FUNCTION_BLOCK Q_SoftKeyMask (* Command change soft key mask( Part 6 - F.36 ) *)
  (* Standard: ISO 11783-6; Description: Copyright (c) 2022 HR Agrartechnik GmbH This program and the accompanying materials are made available under the terms of the Eclipse Public License 2.0 which is available at https://www.eclipse.org/legal/epl-2.0/ SPDX-License-Identifier: EPL-2.0 see Description Tab *)
  (* Version 1.0, 2022-07-08, Franz Höpfinger, HR Agrartechnik GmbH *)
  (* Documentation:
  Command change soft key mask( Part 6 - F.36 )
   This command is used to change the soft key mask associated with a data or alarm mask object.
   param[in] {type, uint8_t}
   1 == Data, 2 == Alarm
   param[in] {dataOrAlarmMaskObjectID, uint16_t}
   Object ID of active Mask
   param[in] {newSoftKeyMaskObjectID, uint16_t}
   Object ID of (new) soft key mask
   Return Values: 
   int16_t
    - VT_E_NO_ERR (0) - OK
   - VT_E_OVERFLOW (-6) - buffer overflow
   - VT_E_NOACT (-8) - Command not possible in current state
   - VT_E_NO_INSTANCE (-21) - No VT client available
   - VT_E_ISO_INSTANCE_INVALID (-129) - Identifier for instance (connection) invalid
   - VT_E_NOT_ALIVE (-130) - Identifier for instance valid, but VT Dead.
  *)
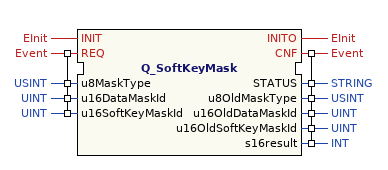
  EVENT_INPUT
    INIT : EInit; (* Service Initialization *)
    REQ WITH u16DataMaskId, u16SoftKeyMaskId, u8MaskType; (* Service Request *)
  END_EVENT
  EVENT_OUTPUT
    INITO : EInit; (* Initialization Confirm *)
    CNF WITH STATUS, s16result, u16OldDataMaskId, u16OldSoftKeyMaskId, u8OldMaskType; (* Confirmation of Requested Service *)
  END_EVENT
  VAR_INPUT
    u8MaskType : USINT; (* 1 == Data, 2 == Alarm *)
    u16DataMaskId : UINT; (* Object ID of active Mask *)
    u16SoftKeyMaskId : UINT; (* Object ID of (new) soft key mask *)
  END_VAR
  VAR_OUTPUT
    STATUS : STRING; (* Service Status *)
    u8OldMaskType : USINT;
    u16OldDataMaskId : UINT; (* Old object ID of active Mask *)
    u16OldSoftKeyMaskId : UINT; (* Old object ID of (new) soft key mask *)
    s16result : INT; (* retval see description *)
  END_VAR
END_FUNCTION_BLOCK
